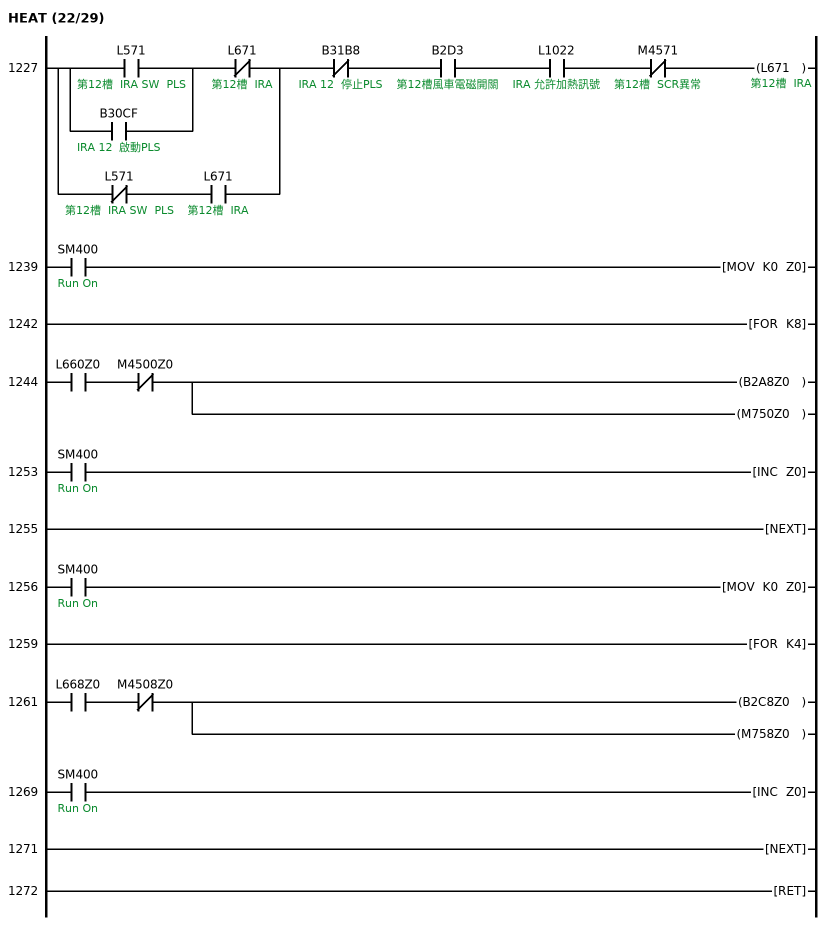
[picture p168: ladder of HEAT, rungs at steps 1227 to 1272]
1227  LD      L571  ; 第12槽  IRA SW  PLS
      OR      B30CF  ; IRA 12  啟動PLS
      ANI     L671  ; 第12槽  IRA
      LDI     L571  ; 第12槽  IRA SW  PLS
      AND     L671  ; 第12槽  IRA
      ORB
      ANI     B31B8  ; IRA 12  停止PLS
      AND     B2D3  ; 第12槽風車電磁開關
      AND     L1022  ; IRA 允許加熱訊號
      ANI     M4571  ; 第12槽  SCR異常
      OUT     L671  ; 第12槽  IRA
1239  LD      SM400  ; Run On
      MOV     K0 Z0
1242  FOR     K8
1244  LD      L660Z0
      ANI     M4500Z0
      OUT     B2A8Z0
      OUT     M750Z0
1253  LD      SM400  ; Run On
      INC     Z0
1255  NEXT
1256  LD      SM400  ; Run On
      MOV     K0 Z0
1259  FOR     K4
1261  LD      L668Z0
      ANI     M4508Z0
      OUT     B2C8Z0
      OUT     M758Z0
1269  LD      SM400  ; Run On
      INC     Z0
1271  NEXT
1272  RET
      P450
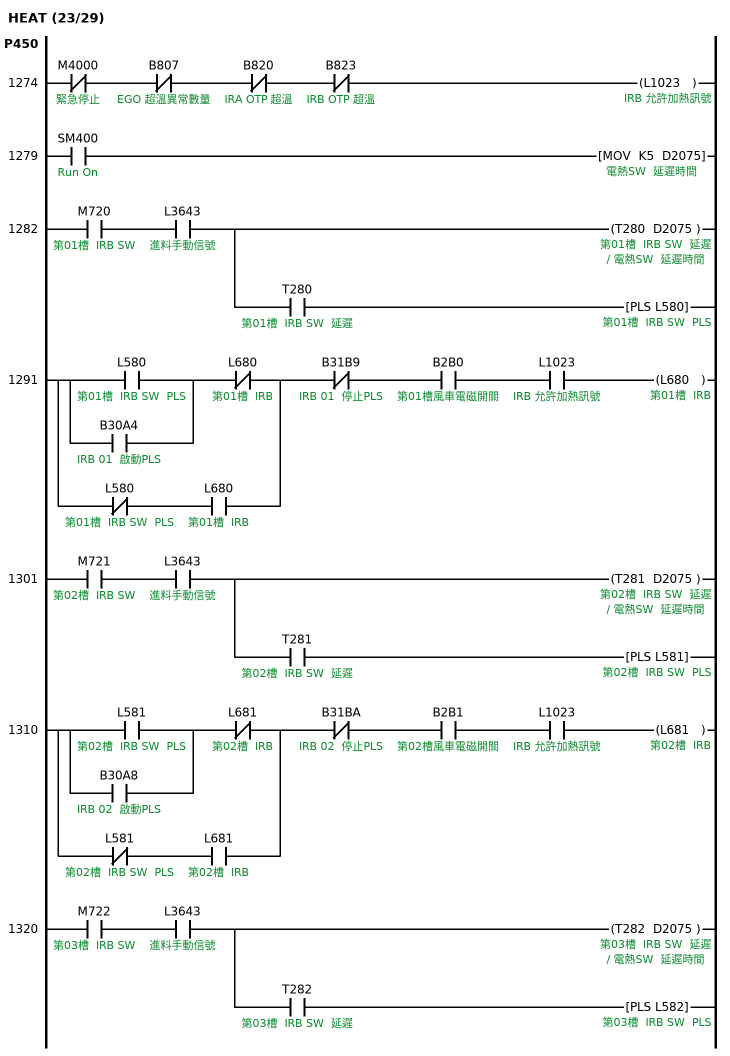
1274  LDI     M4000  ; 緊急停止
      ANI     B807  ; EGO 超溫異常數量
      ANI     B820  ; IRA OTP 超溫
      ANI     B823  ; IRB OTP 超溫
      OUT     L1023  ; IRB 允許加熱訊號
1279  LD      SM400  ; Run On
      MOV     K5 D2075
1282  LD      M720  ; 第01槽  IRB SW
      AND     L3643  ; 進料手動信號
      OUT     T280 D2075  ; 第01槽  IRB SW  延遲 / 電熱SW  延遲時間
      AND     T280  ; 第01槽  IRB SW  延遲
      PLS     L580  ; 第01槽  IRB SW  PLS
1291  LD      L580  ; 第01槽  IRB SW  PLS
      OR      B30A4  ; IRB 01  啟動PLS
      ANI     L680  ; 第01槽  IRB
      LDI     L580  ; 第01槽  IRB SW  PLS
      AND     L680  ; 第01槽  IRB
      ORB
      ANI     B31B9  ; IRB 01  停止PLS
      AND     B2B0  ; 第01槽風車電磁開關
      AND     L1023  ; IRB 允許加熱訊號
      OUT     L680  ; 第01槽  IRB
1301  LD      M721  ; 第02槽  IRB SW
      AND     L3643  ; 進料手動信號
      OUT     T281 D2075  ; 第02槽  IRB SW  延遲 / 電熱SW  延遲時間
      AND     T281  ; 第02槽  IRB SW  延遲
      PLS     L581  ; 第02槽  IRB SW  PLS
1310  LD      L581  ; 第02槽  IRB SW  PLS
      OR      B30A8  ; IRB 02  啟動PLS
      ANI     L681  ; 第02槽  IRB
      LDI     L581  ; 第02槽  IRB SW  PLS
      AND     L681  ; 第02槽  IRB
      ORB
      ANI     B31BA  ; IRB 02  停止PLS
      AND     B2B1  ; 第02槽風車電磁開關
      AND     L1023  ; IRB 允許加熱訊號
      OUT     L681  ; 第02槽  IRB
1320  LD      M722  ; 第03槽  IRB SW
      AND     L3643  ; 進料手動信號
      OUT     T282 D2075  ; 第03槽  IRB SW  延遲 / 電熱SW  延遲時間
      AND     T282  ; 第03槽  IRB SW  延遲
      PLS     L582  ; 第03槽  IRB SW  PLS
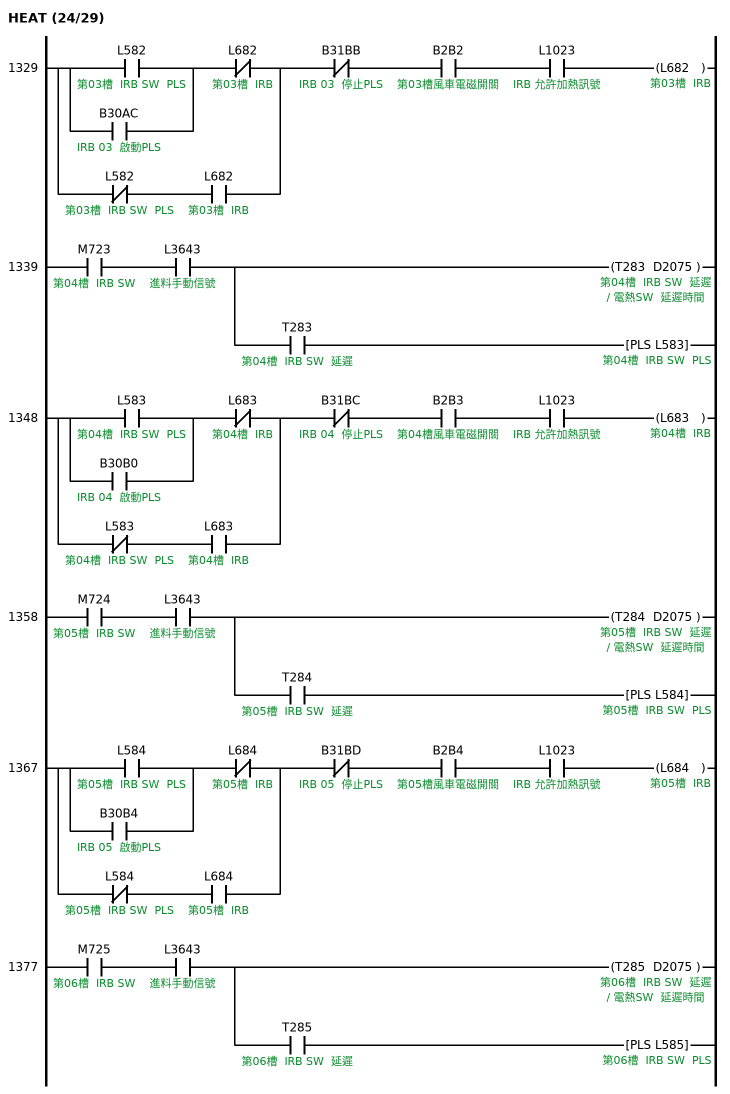
1329  LD      L582  ; 第03槽  IRB SW  PLS
      OR      B30AC  ; IRB 03  啟動PLS
      ANI     L682  ; 第03槽  IRB
      LDI     L582  ; 第03槽  IRB SW  PLS
      AND     L682  ; 第03槽  IRB
      ORB
      ANI     B31BB  ; IRB 03  停止PLS
      AND     B2B2  ; 第03槽風車電磁開關
      AND     L1023  ; IRB 允許加熱訊號
      OUT     L682  ; 第03槽  IRB
1339  LD      M723  ; 第04槽  IRB SW
      AND     L3643  ; 進料手動信號
      OUT     T283 D2075  ; 第04槽  IRB SW  延遲 / 電熱SW  延遲時間
      AND     T283  ; 第04槽  IRB SW  延遲
      PLS     L583  ; 第04槽  IRB SW  PLS
1348  LD      L583  ; 第04槽  IRB SW  PLS
      OR      B30B0  ; IRB 04  啟動PLS
      ANI     L683  ; 第04槽  IRB
      LDI     L583  ; 第04槽  IRB SW  PLS
      AND     L683  ; 第04槽  IRB
      ORB
      ANI     B31BC  ; IRB 04  停止PLS
      AND     B2B3  ; 第04槽風車電磁開關
      AND     L1023  ; IRB 允許加熱訊號
      OUT     L683  ; 第04槽  IRB
1358  LD      M724  ; 第05槽  IRB SW
      AND     L3643  ; 進料手動信號
      OUT     T284 D2075  ; 第05槽  IRB SW  延遲 / 電熱SW  延遲時間
      AND     T284  ; 第05槽  IRB SW  延遲
      PLS     L584  ; 第05槽  IRB SW  PLS
1367  LD      L584  ; 第05槽  IRB SW  PLS
      OR      B30B4  ; IRB 05  啟動PLS
      ANI     L684  ; 第05槽  IRB
      LDI     L584  ; 第05槽  IRB SW  PLS
      AND     L684  ; 第05槽  IRB
      ORB
      ANI     B31BD  ; IRB 05  停止PLS
      AND     B2B4  ; 第05槽風車電磁開關
      AND     L1023  ; IRB 允許加熱訊號
      OUT     L684  ; 第05槽  IRB
1377  LD      M725  ; 第06槽  IRB SW
      AND     L3643  ; 進料手動信號
      OUT     T285 D2075  ; 第06槽  IRB SW  延遲 / 電熱SW  延遲時間
      AND     T285  ; 第06槽  IRB SW  延遲
      PLS     L585  ; 第06槽  IRB SW  PLS
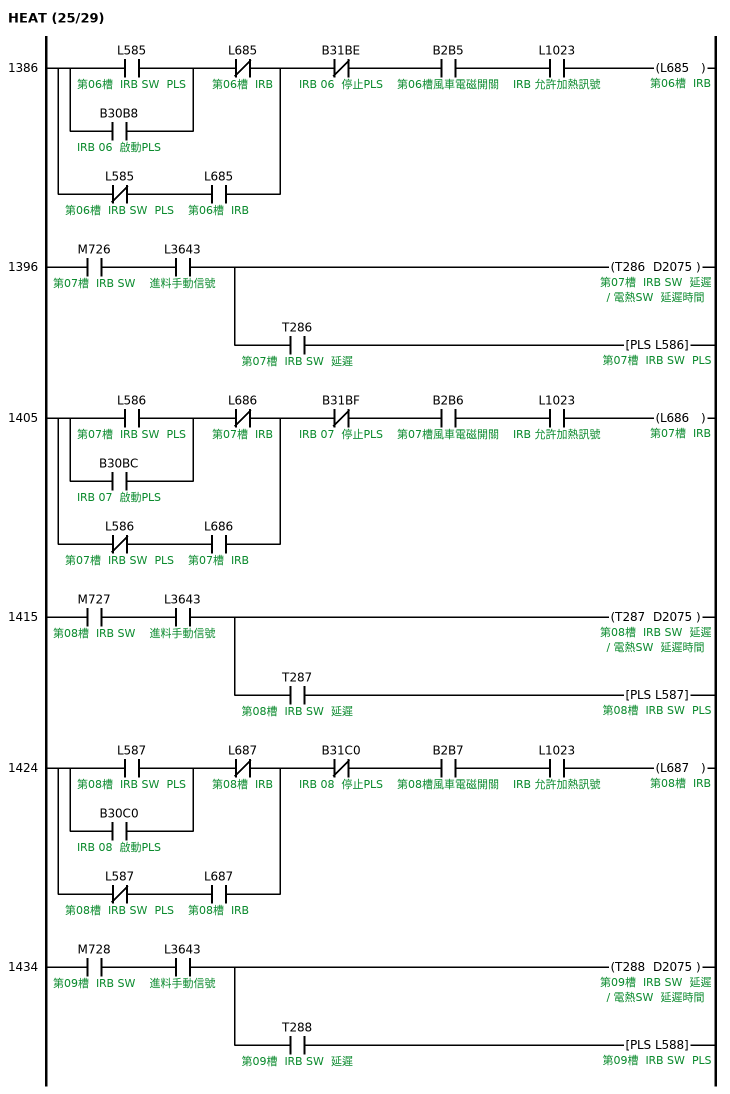
1386  LD      L585  ; 第06槽  IRB SW  PLS
      OR      B30B8  ; IRB 06  啟動PLS
      ANI     L685  ; 第06槽  IRB
      LDI     L585  ; 第06槽  IRB SW  PLS
      AND     L685  ; 第06槽  IRB
      ORB
      ANI     B31BE  ; IRB 06  停止PLS
      AND     B2B5  ; 第06槽風車電磁開關
      AND     L1023  ; IRB 允許加熱訊號
      OUT     L685  ; 第06槽  IRB
1396  LD      M726  ; 第07槽  IRB SW
      AND     L3643  ; 進料手動信號
      OUT     T286 D2075  ; 第07槽  IRB SW  延遲 / 電熱SW  延遲時間
      AND     T286  ; 第07槽  IRB SW  延遲
      PLS     L586  ; 第07槽  IRB SW  PLS
1405  LD      L586  ; 第07槽  IRB SW  PLS
      OR      B30BC  ; IRB 07  啟動PLS
      ANI     L686  ; 第07槽  IRB
      LDI     L586  ; 第07槽  IRB SW  PLS
      AND     L686  ; 第07槽  IRB
      ORB
      ANI     B31BF  ; IRB 07  停止PLS
      AND     B2B6  ; 第07槽風車電磁開關
      AND     L1023  ; IRB 允許加熱訊號
      OUT     L686  ; 第07槽  IRB
1415  LD      M727  ; 第08槽  IRB SW
      AND     L3643  ; 進料手動信號
      OUT     T287 D2075  ; 第08槽  IRB SW  延遲 / 電熱SW  延遲時間
      AND     T287  ; 第08槽  IRB SW  延遲
      PLS     L587  ; 第08槽  IRB SW  PLS
1424  LD      L587  ; 第08槽  IRB SW  PLS
      OR      B30C0  ; IRB 08  啟動PLS
      ANI     L687  ; 第08槽  IRB
      LDI     L587  ; 第08槽  IRB SW  PLS
      AND     L687  ; 第08槽  IRB
      ORB
      ANI     B31C0  ; IRB 08  停止PLS
      AND     B2B7  ; 第08槽風車電磁開關
      AND     L1023  ; IRB 允許加熱訊號
      OUT     L687  ; 第08槽  IRB
1434  LD      M728  ; 第09槽  IRB SW
      AND     L3643  ; 進料手動信號
      OUT     T288 D2075  ; 第09槽  IRB SW  延遲 / 電熱SW  延遲時間
      AND     T288  ; 第09槽  IRB SW  延遲
      PLS     L588  ; 第09槽  IRB SW  PLS
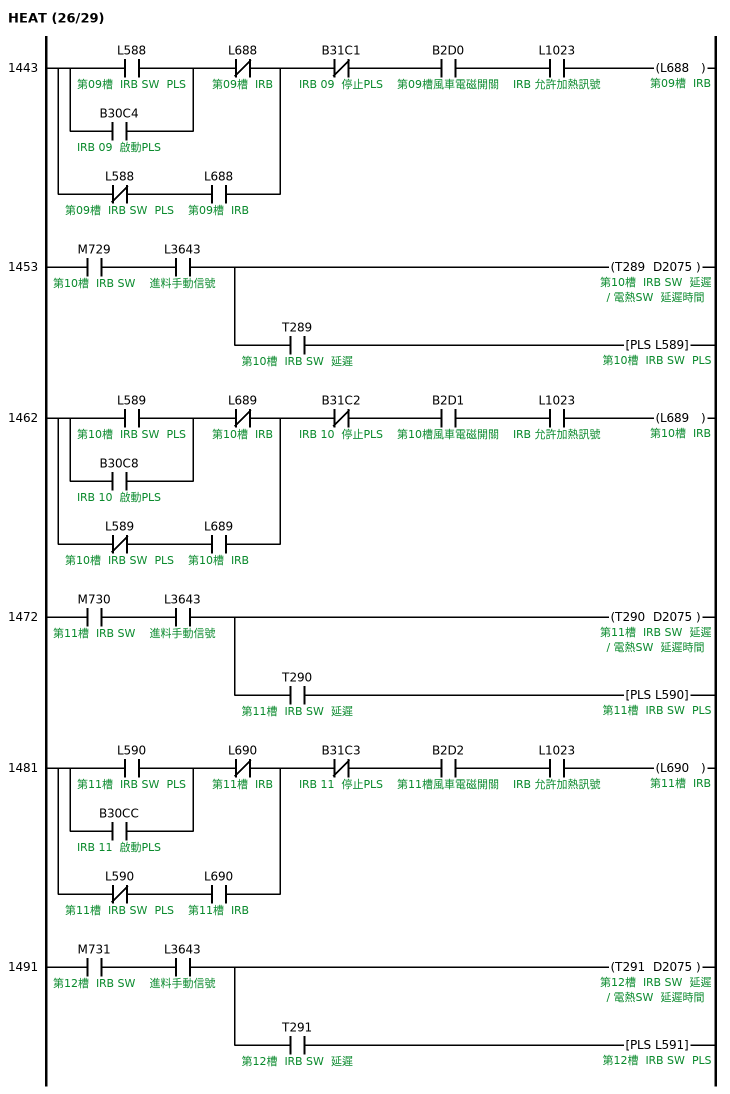
1443  LD      L588  ; 第09槽  IRB SW  PLS
      OR      B30C4  ; IRB 09  啟動PLS
      ANI     L688  ; 第09槽  IRB
      LDI     L588  ; 第09槽  IRB SW  PLS
      AND     L688  ; 第09槽  IRB
      ORB
      ANI     B31C1  ; IRB 09  停止PLS
      AND     B2D0  ; 第09槽風車電磁開關
      AND     L1023  ; IRB 允許加熱訊號
      OUT     L688  ; 第09槽  IRB
1453  LD      M729  ; 第10槽  IRB SW
      AND     L3643  ; 進料手動信號
      OUT     T289 D2075  ; 第10槽  IRB SW  延遲 / 電熱SW  延遲時間
      AND     T289  ; 第10槽  IRB SW  延遲
      PLS     L589  ; 第10槽  IRB SW  PLS
1462  LD      L589  ; 第10槽  IRB SW  PLS
      OR      B30C8  ; IRB 10  啟動PLS
      ANI     L689  ; 第10槽  IRB
      LDI     L589  ; 第10槽  IRB SW  PLS
      AND     L689  ; 第10槽  IRB
      ORB
      ANI     B31C2  ; IRB 10  停止PLS
      AND     B2D1  ; 第10槽風車電磁開關
      AND     L1023  ; IRB 允許加熱訊號
      OUT     L689  ; 第10槽  IRB
1472  LD      M730  ; 第11槽  IRB SW
      AND     L3643  ; 進料手動信號
      OUT     T290 D2075  ; 第11槽  IRB SW  延遲 / 電熱SW  延遲時間
      AND     T290  ; 第11槽  IRB SW  延遲
      PLS     L590  ; 第11槽  IRB SW  PLS
1481  LD      L590  ; 第11槽  IRB SW  PLS
      OR      B30CC  ; IRB 11  啟動PLS
      ANI     L690  ; 第11槽  IRB
      LDI     L590  ; 第11槽  IRB SW  PLS
      AND     L690  ; 第11槽  IRB
      ORB
      ANI     B31C3  ; IRB 11  停止PLS
      AND     B2D2  ; 第11槽風車電磁開關
      AND     L1023  ; IRB 允許加熱訊號
      OUT     L690  ; 第11槽  IRB
1491  LD      M731  ; 第12槽  IRB SW
      AND     L3643  ; 進料手動信號
      OUT     T291 D2075  ; 第12槽  IRB SW  延遲 / 電熱SW  延遲時間
      AND     T291  ; 第12槽  IRB SW  延遲
      PLS     L591  ; 第12槽  IRB SW  PLS
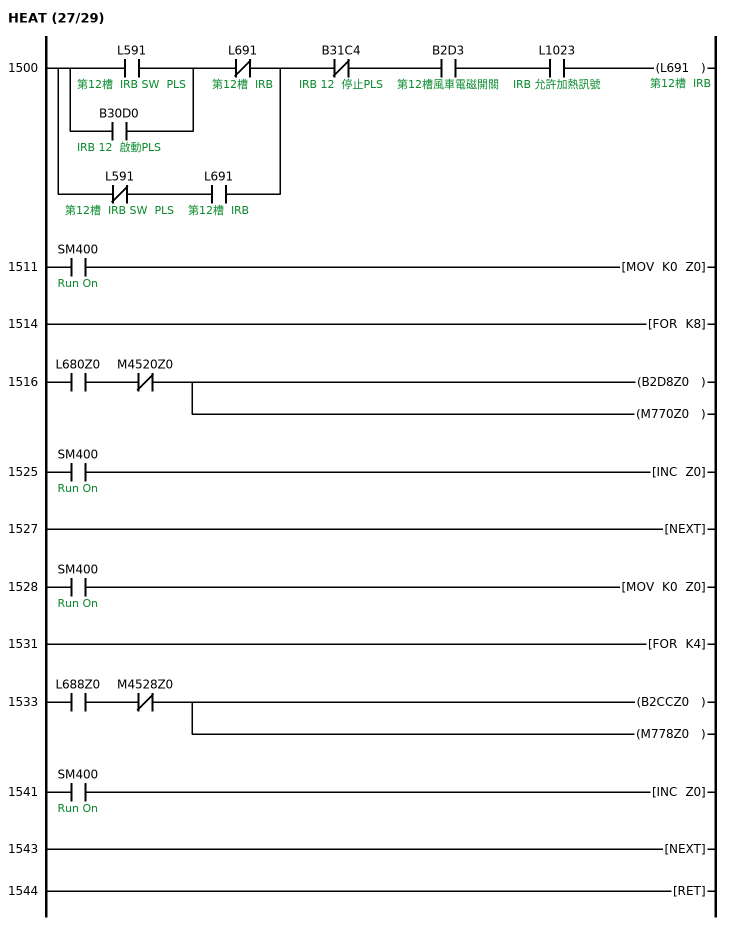
1500  LD      L591  ; 第12槽  IRB SW  PLS
      OR      B30D0  ; IRB 12  啟動PLS
      ANI     L691  ; 第12槽  IRB
      LDI     L591  ; 第12槽  IRB SW  PLS
      AND     L691  ; 第12槽  IRB
      ORB
      ANI     B31C4  ; IRB 12  停止PLS
      AND     B2D3  ; 第12槽風車電磁開關
      AND     L1023  ; IRB 允許加熱訊號
      OUT     L691  ; 第12槽  IRB
1511  LD      SM400  ; Run On
      MOV     K0 Z0
1514  FOR     K8
1516  LD      L680Z0
      ANI     M4520Z0
      OUT     B2D8Z0
      OUT     M770Z0
1525  LD      SM400  ; Run On
      INC     Z0
1527  NEXT
1528  LD      SM400  ; Run On
      MOV     K0 Z0
1531  FOR     K4
1533  LD      L688Z0
      ANI     M4528Z0
      OUT     B2CCZ0
      OUT     M778Z0
1541  LD      SM400  ; Run On
      INC     Z0
1543  NEXT
1544  RET
; /* Length=每段爐體長度_Section=爐體段數 */
      P460
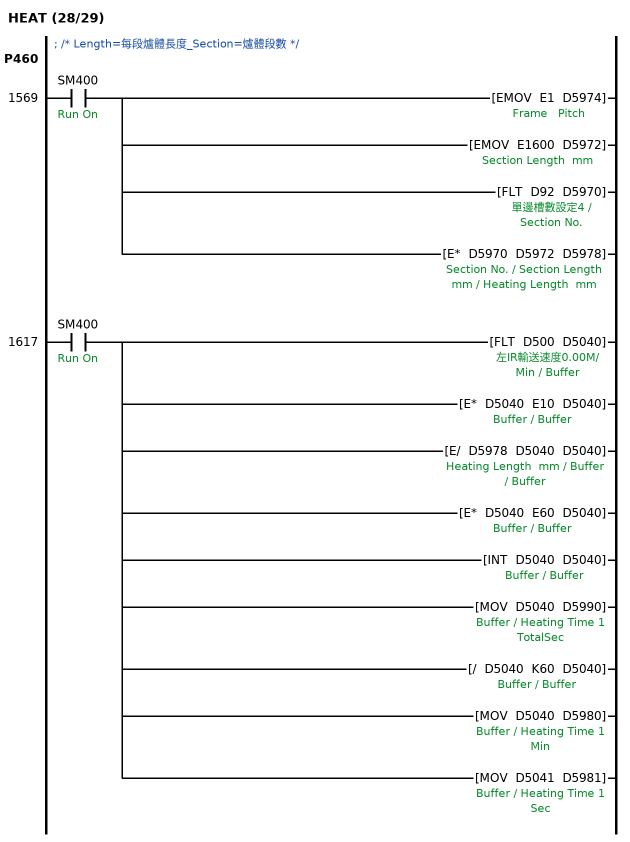
1569  LD      SM400  ; Run On
      EMOV    E1 D5974  ; Frame   Pitch
      EMOV    E1600 D5972  ; Section Length  mm
        [note] /* 加熱爐體每段長度mm */
      FLT     D92 D5970  ; 單邊槽數設定4 / Section No.
        [note] /* 加熱段數 */
      E*      D5970 D5972 D5978  ; Heating Length  mm
        [note] /* 加熱段_總長度mm */
1617  LD      SM400  ; Run On
      FLT     D500 D5040  ; 左IR輸送速度0.00M/Min / Buffer
      E*      D5040 E10 D5040
      E/      D5978 D5040 D5040
        [note] / 板子經過爐體總時間_E0.000Min /
      E*      D5040 E60 D5040
        [note] / 板子經過爐體總時間_E0.000Sec /
      INT     D5040 D5040
      MOV     D5040 D5990  ; Heating Time 1  TotalSec
      /       D5040 K60 D5040
      MOV     D5040 D5980  ; Heating Time 1  Min
      MOV     D5041 D5981  ; Buffer / Heating Time 1  Sec
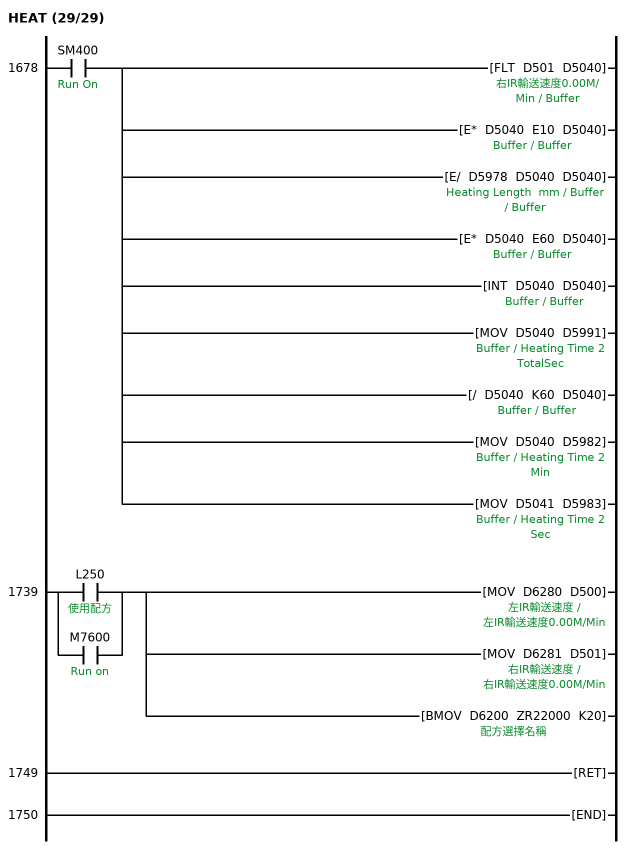
1678  LD      SM400  ; Run On
      FLT     D501 D5040  ; 右IR輸送速度0.00M/Min
      E*      D5040 E10 D5040
      E/      D5978 D5040 D5040
        [note] / 板子經過爐體總時間_E0.000Min /
      E*      D5040 E60 D5040
        [note] / 板子經過爐體總時間_E0.000Sec /
      INT     D5040 D5040
      MOV     D5040 D5991  ; Heating Time 2  TotalSec
      /       D5040 K60 D5040
      MOV     D5040 D5982  ; Heating Time 2  Min
      MOV     D5041 D5983  ; Heating Time 2  Sec
1739  LD      L250  ; 使用配方
      OR      M7600  ; Run on
      MOV     D6280 D500  ; 左IR輸送速度
      MOV     D6281 D501  ; 右IR輸送速度
      BMOV    D6200 ZR22000 K20  ; 配方選擇名稱
1749  RET
1750  END
END_PROGRAM

PROGRAM ALARM
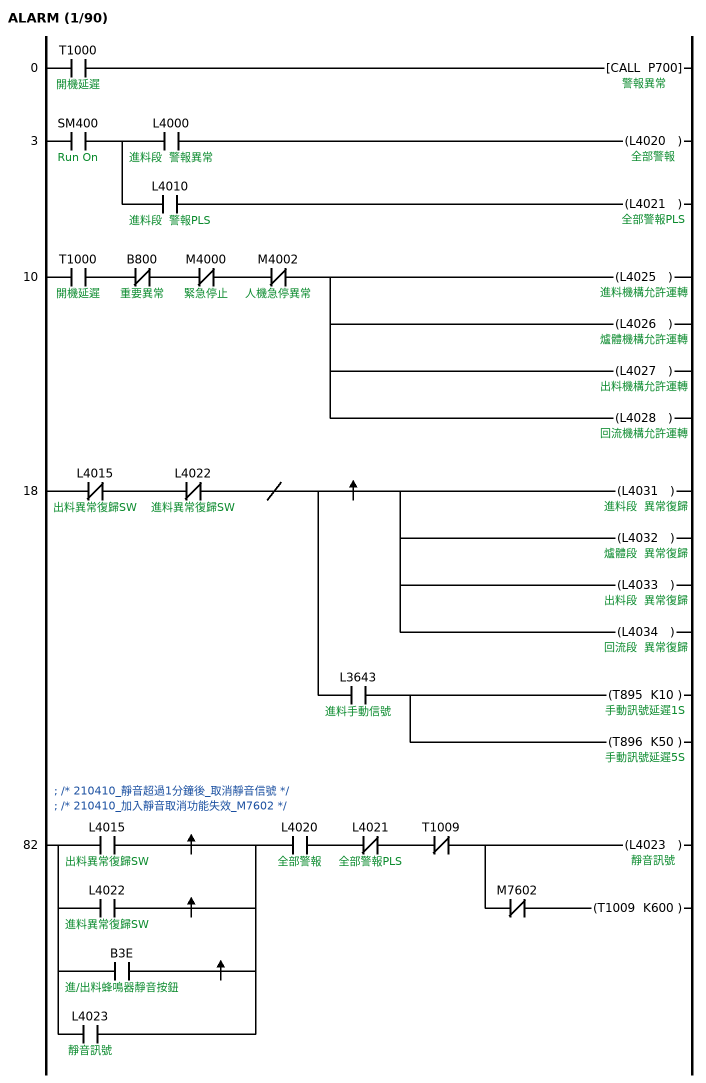
0     LD      T1000  ; 開機延遲
      CALL    P700  ; 警報異常
3     LD      SM400  ; Run On
      MPS
      AND     L4000  ; 進料段  警報異常
      OUT     L4020  ; 全部警報
      MPP
      AND     L4010  ; 進料段  警報PLS
      OUT     L4021  ; 全部警報PLS
10    LD      T1000  ; 開機延遲
      ANI     B800  ; 重要異常
      ANI     M4000  ; 緊急停止
      ANI     M4002  ; 人機急停異常
      OUT     L4025  ; 進料機構允許運轉
      OUT     L4026  ; 爐體機構允許運轉
      OUT     L4027  ; 出料機構允許運轉
      OUT     L4028  ; 回流機構允許運轉
18    LDI     L4015  ; 出料異常復歸SW
      ANI     L4022  ; 進料異常復歸SW
      INV
      MPS
      MEP
      OUT     L4031  ; 進料段  異常復歸
      OUT     L4032  ; 爐體段  異常復歸
      OUT     L4033  ; 出料段  異常復歸
      OUT     L4034  ; 回流段  異常復歸
      MPP
      AND     L3643  ; 進料手動信號
      OUT     T895 K10  ; 手動訊號延遲1S
      OUT     T896 K50  ; 手動訊號延遲5S
; /* 210410_靜音超過1分鐘後_取消靜音信號 */
; /* 210410_加入靜音取消功能失效_M7602 */
82    LD      L4015  ; 出料異常復歸SW
      MEP
      LD      L4022  ; 進料異常復歸SW
      MEP
      ORB
      LD      B3E  ; 進/出料蜂鳴器靜音按鈕
      MEP
      ORB
      OR      L4023  ; 靜音訊號
      AND     L4020  ; 全部警報
      ANI     L4021  ; 全部警報PLS
      ANI     T1009
      OUT     L4023  ; 靜音訊號
      ANI     M7602
      OUT     T1009 K600
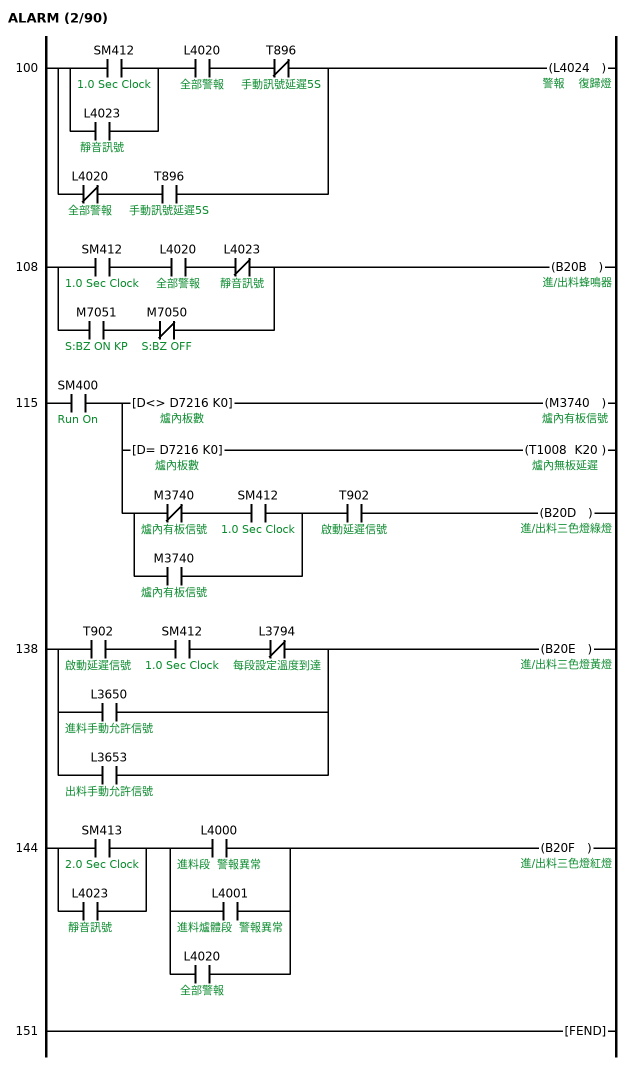
100   LD      SM412  ; 1.0 Sec Clock
      OR      L4023  ; 靜音訊號
      AND     L4020  ; 全部警報
      ANI     T896  ; 手動訊號延遲5S
      LDI     L4020  ; 全部警報
      AND     T896  ; 手動訊號延遲5S
      ORB
      OUT     L4024  ; 警報    復歸燈
108   LD      SM412  ; 1.0 Sec Clock
      AND     L4020  ; 全部警報
      ANI     L4023  ; 靜音訊號
      LD      M7051  ; S:BZ ON KP
      ANI     M7050  ; S:BZ OFF
      ORB
      OUT     B20B  ; 進/出料蜂鳴器
115   LD      SM400  ; Run On
      MPS
      ANDD<>  D7216 K0  ; 爐內板數
      OUT     M3740  ; 爐內有板信號
      MRD
      ANDD=   D7216 K0  ; 爐內板數
      OUT     T1008 K20  ; 爐內無板延遲
      MPP
      LDI     M3740  ; 爐內有板信號
      AND     SM412  ; 1.0 Sec Clock
      OR      M3740  ; 爐內有板信號
      ANB
      AND     T902  ; 啟動延遲信號
      OUT     B20D  ; 進/出料三色燈綠燈
138   LD      T902  ; 啟動延遲信號
      AND     SM412  ; 1.0 Sec Clock
      ANI     L3794  ; 每段設定溫度到達
      OR      L3650  ; 進料手動允許信號
      OR      L3653  ; 出料手動允許信號
      OUT     B20E  ; 進/出料三色燈黃燈
144   LD      SM413  ; 2.0 Sec Clock
      OR      L4023  ; 靜音訊號
      LD      L4000  ; 進料段  警報異常
      OR      L4001  ; 進料爐體段  警報異常
      OR      L4020  ; 全部警報
      ANB
      OUT     B20F  ; 進/出料三色燈紅燈
151   FEND
      P700
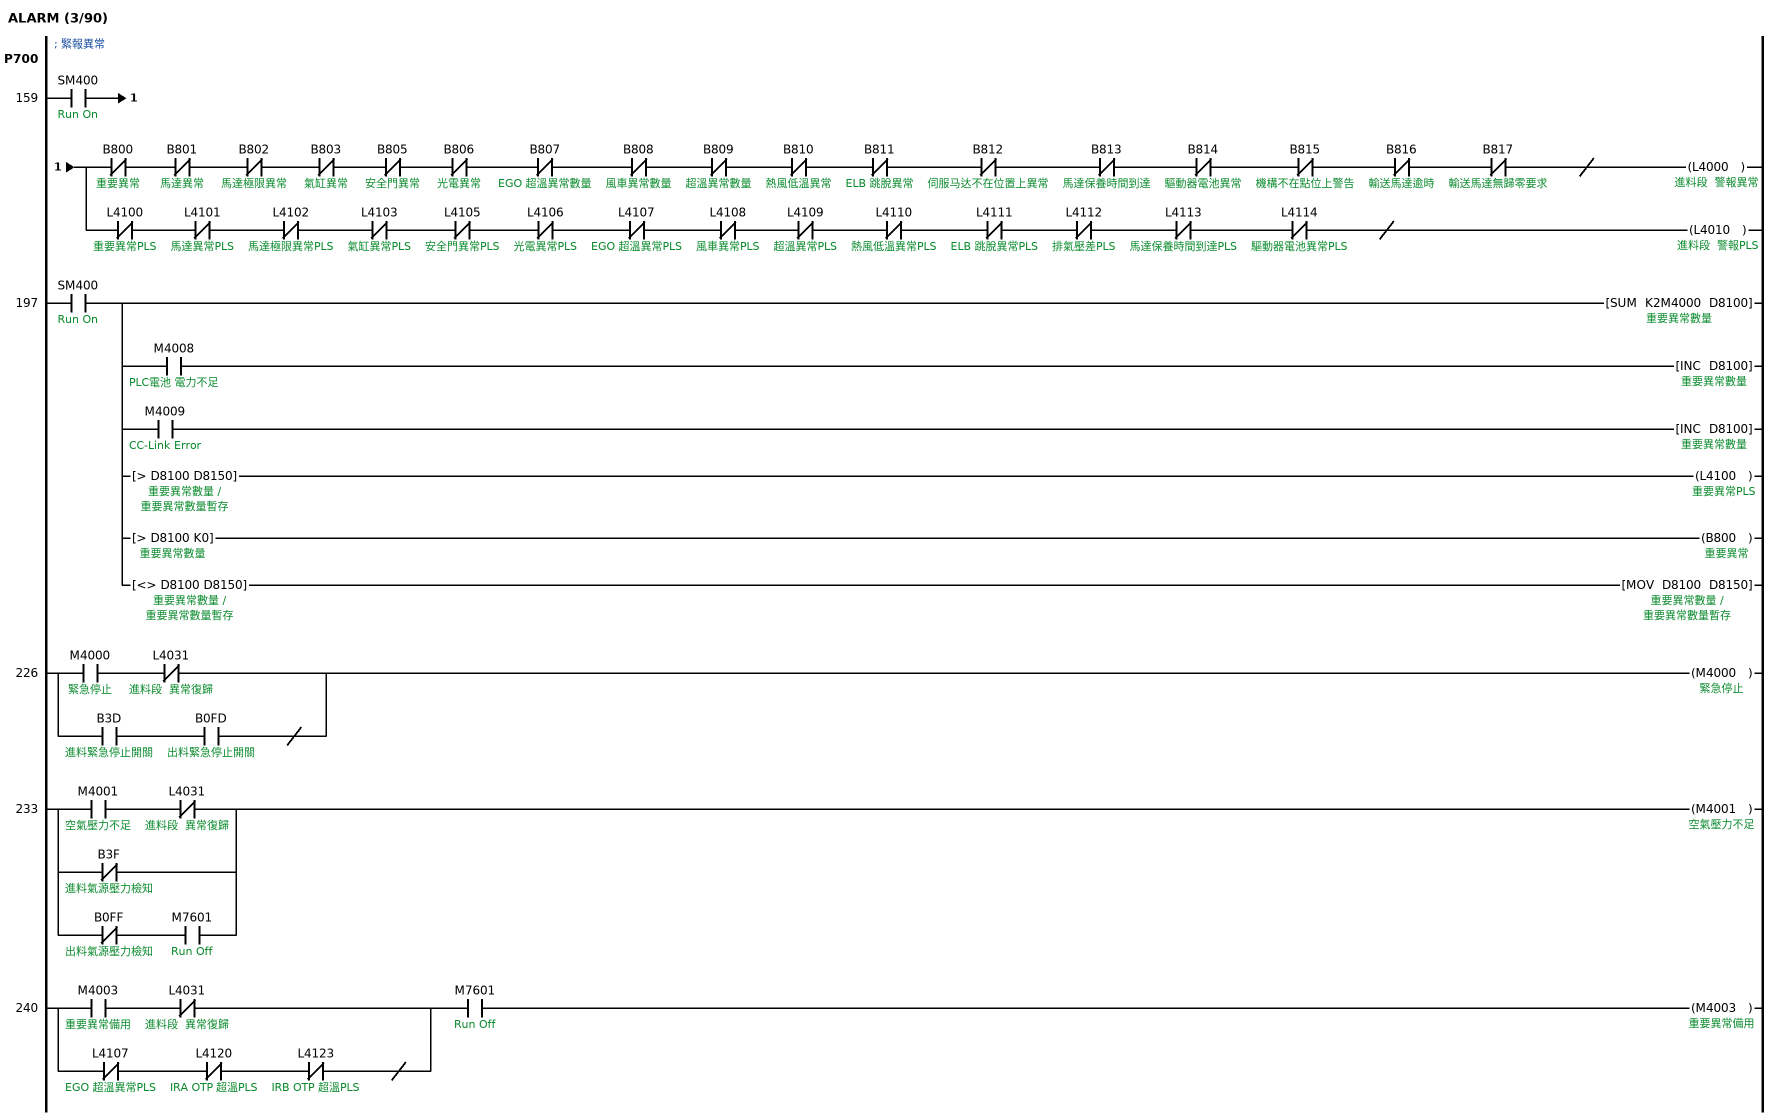
; 緊報異常
159   LD      SM400  ; Run On
      MPS
      ANI     B800  ; 重要異常
      ANI     B801  ; 馬達異常
      ANI     B802  ; 馬達極限異常
      ANI     B803  ; 氣缸異常
      ANI     B805  ; 安全門異常
      ANI     B806  ; 光電異常
      ANI     B807  ; EGO 超溫異常數量
      ANI     B808  ; 風車異常數量
      ANI     B809  ; 超溫異常數量
      ANI     B810  ; 熱風低溫異常
      ANI     B811  ; ELB 跳脫異常
      ANI     B812  ; 伺服马达不在位置上異常
      ANI     B813  ; 馬達保養時間到達
      ANI     B814  ; 驅動器電池異常
      ANI     B815  ; 機構不在點位上警告
      ANI     B816  ; 輸送馬達逾時
      ANI     B817  ; 輸送馬達無歸零要求
      INV
      OUT     L4000  ; 進料段  警報異常
      MPP
      ANI     L4100  ; 重要異常PLS
      ANI     L4101  ; 馬達異常PLS
      ANI     L4102  ; 馬達極限異常PLS
      ANI     L4103  ; 氣缸異常PLS
      ANI     L4105  ; 安全門異常PLS
      ANI     L4106  ; 光電異常PLS
      ANI     L4107  ; EGO 超溫異常PLS
      ANI     L4108  ; 風車異常PLS
      ANI     L4109  ; 超溫異常PLS
      ANI     L4110  ; 熱風低溫異常PLS
      ANI     L4111  ; ELB 跳脫異常PLS
      ANI     L4112  ; 排氣壓差PLS
      ANI     L4113  ; 馬達保養時間到達PLS
      ANI     L4114  ; 驅動器電池異常PLS
      INV
      OUT     L4010  ; 進料段  警報PLS
197   LD      SM400  ; Run On
      SUM     K2M4000 D8100  ; 重要異常數量
      MPS
      AND     M4008  ; PLC電池 電力不足
      INC     D8100
      MRD
      AND     M4009  ; CC-Link Error
      INC     D8100
      MRD
      AND>    D8100 D8150  ; 重要異常數量 / 重要異常數量暫存
      OUT     L4100  ; 重要異常PLS
      MRD
      AND>    D8100 K0  ; 重要異常數量
      OUT     B800  ; 重要異常
      MPP
      AND<>   D8100 D8150  ; 重要異常數量 / 重要異常數量暫存
      MOV     D8100 D8150
226   LD      M4000  ; 緊急停止
      ANI     L4031  ; 進料段  異常復歸
      LD      B3D  ; 進料緊急停止開關
      AND     B0FD  ; 出料緊急停止開關
      INV
      ORB
      OUT     M4000  ; 緊急停止
233   LD      M4001  ; 空氣壓力不足
      ANI     L4031  ; 進料段  異常復歸
      ORI     B3F  ; 進料氣源壓力檢知
      LDI     B0FF  ; 出料氣源壓力檢知
      AND     M7601  ; Run Off
      ORB
      OUT     M4001  ; 空氣壓力不足
240   LD      M4003  ; 重要異常備用
      ANI     L4031  ; 進料段  異常復歸
      LDI     L4107  ; EGO 超溫異常PLS
      ANI     L4120  ; IRA OTP 超溫PLS
      ANI     L4123  ; IRB OTP 超溫PLS
      INV
      ORB
      AND     M7601  ; Run Off
      OUT     M4003  ; 重要異常備用
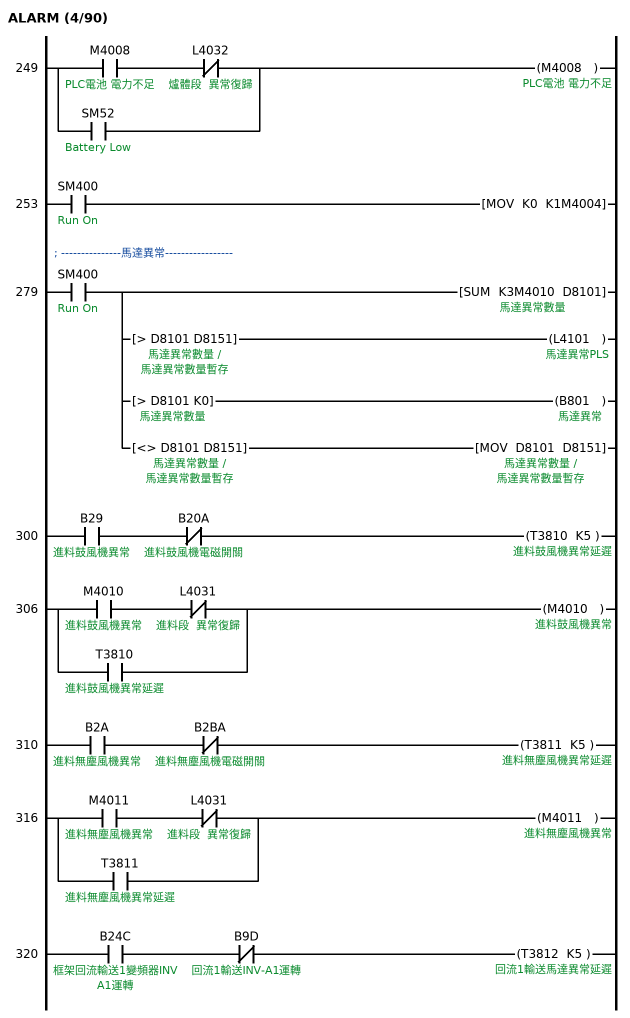
249   LD      M4008  ; PLC電池 電力不足
      ANI     L4032  ; 爐體段  異常復歸
      OR      SM52  ; Battery Low
      OUT     M4008  ; PLC電池 電力不足
253   LD      SM400  ; Run On
      MOV     K0 K1M4004  ; 重要異常備用
; ---------------馬達異常-----------------
279   LD      SM400  ; Run On
      SUM     K3M4010 D8101  ; 進料鼓風機異常 / 馬達異常數量
      MPS
      AND>    D8101 D8151  ; 馬達異常數量 / 馬達異常數量暫存
      OUT     L4101  ; 馬達異常PLS
      MRD
      AND>    D8101 K0  ; 馬達異常數量
      OUT     B801  ; 馬達異常
      MPP
      AND<>   D8101 D8151  ; 馬達異常數量 / 馬達異常數量暫存
      MOV     D8101 D8151
300   LD      B29  ; 進料鼓風機異常
      ANI     B20A  ; 進料鼓風機電磁開關
      OUT     T3810 K5  ; 進料鼓風機異常延遲
306   LD      M4010  ; 進料鼓風機異常
      ANI     L4031  ; 進料段  異常復歸
      OR      T3810  ; 進料鼓風機異常延遲
      OUT     M4010  ; 進料鼓風機異常
310   LD      B2A  ; 進料無塵風機異常
      ANI     B2BA  ; 進料無塵風機電磁開關
      OUT     T3811 K5  ; 進料無塵風機異常延遲
316   LD      M4011  ; 進料無塵風機異常
      ANI     L4031  ; 進料段  異常復歸
      OR      T3811  ; 進料無塵風機異常延遲
      OUT     M4011  ; 進料無塵風機異常
320   LD      B24C  ; 框架回流輸送1變頻器INVA1運轉
      ANI     B9D  ; 回流1輸送INV-A1運轉
      OUT     T3812 K5  ; 回流1輸送馬達異常延遲
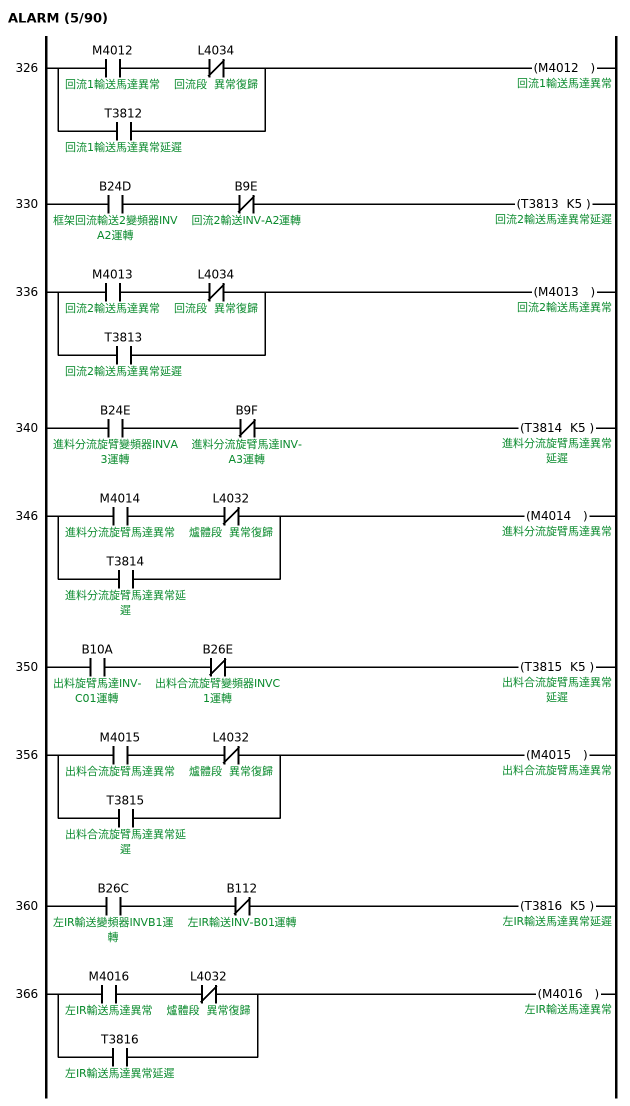
326   LD      M4012  ; 回流1輸送馬達異常
      ANI     L4034  ; 回流段  異常復歸
      OR      T3812  ; 回流1輸送馬達異常延遲
      OUT     M4012  ; 回流1輸送馬達異常
330   LD      B24D  ; 框架回流輸送2變頻器INVA2運轉
      ANI     B9E  ; 回流2輸送INV-A2運轉
      OUT     T3813 K5  ; 回流2輸送馬達異常延遲
336   LD      M4013  ; 回流2輸送馬達異常
      ANI     L4034  ; 回流段  異常復歸
      OR      T3813  ; 回流2輸送馬達異常延遲
      OUT     M4013  ; 回流2輸送馬達異常
340   LD      B24E  ; 進料分流旋臂變頻器INVA3運轉
      ANI     B9F  ; 進料分流旋臂馬達INV-A3運轉
      OUT     T3814 K5  ; 進料分流旋臂馬達異常延遲
346   LD      M4014  ; 進料分流旋臂馬達異常
      ANI     L4032  ; 爐體段  異常復歸
      OR      T3814  ; 進料分流旋臂馬達異常延遲
      OUT     M4014  ; 進料分流旋臂馬達異常
350   LD      B10A  ; 出料旋臂馬達INV-C01運轉
      ANI     B26E  ; 出料合流旋臂變頻器INVC1運轉
      OUT     T3815 K5  ; 出料合流旋臂馬達異常延遲
356   LD      M4015  ; 出料合流旋臂馬達異常
      ANI     L4032  ; 爐體段  異常復歸
      OR      T3815  ; 出料合流旋臂馬達異常延遲
      OUT     M4015  ; 出料合流旋臂馬達異常
360   LD      B26C  ; 左IR輸送變頻器INVB1運轉
      ANI     B112  ; 左IR輸送INV-B01運轉
      OUT     T3816 K5  ; 左IR輸送馬達異常延遲
366   LD      M4016  ; 左IR輸送馬達異常
      ANI     L4032  ; 爐體段  異常復歸
      OR      T3816  ; 左IR輸送馬達異常延遲
      OUT     M4016  ; 左IR輸送馬達異常
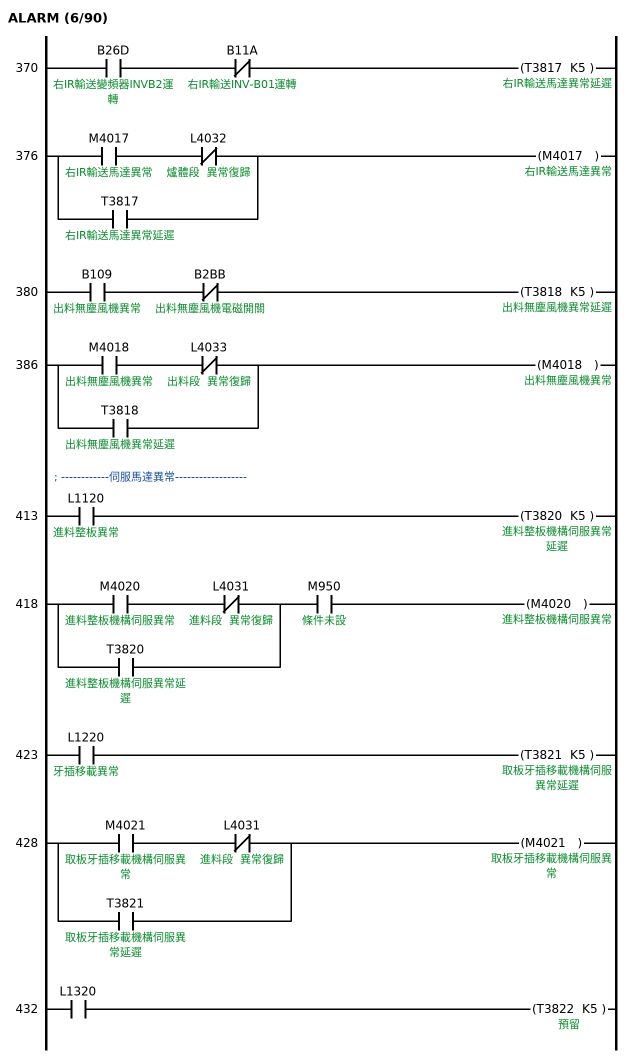
370   LD      B26D  ; 右IR輸送變頻器INVB2運轉
      ANI     B11A  ; 右IR輸送INV-B01運轉
      OUT     T3817 K5  ; 右IR輸送馬達異常延遲
376   LD      M4017  ; 右IR輸送馬達異常
      ANI     L4032  ; 爐體段  異常復歸
      OR      T3817  ; 右IR輸送馬達異常延遲
      OUT     M4017  ; 右IR輸送馬達異常
380   LD      B109  ; 出料無塵風機異常
      ANI     B2BB  ; 出料無塵風機電磁開關
      OUT     T3818 K5  ; 出料無塵風機異常延遲
386   LD      M4018  ; 出料無塵風機異常
      ANI     L4033  ; 出料段  異常復歸
      OR      T3818  ; 出料無塵風機異常延遲
      OUT     M4018  ; 出料無塵風機異常
; ------------伺服馬達異常------------------
413   LD      L1120  ; 進料整板異常
      OUT     T3820 K5  ; 進料整板機構伺服異常延遲
418   LD      M4020  ; 進料整板機構伺服異常
      ANI     L4031  ; 進料段  異常復歸
      OR      T3820  ; 進料整板機構伺服異常延遲
      AND     M950  ; 條件未設
      OUT     M4020  ; 進料整板機構伺服異常
423   LD      L1220  ; 牙插移載異常
      OUT     T3821 K5  ; 取板牙插移載機構伺服異常延遲
428   LD      M4021  ; 取板牙插移載機構伺服異常
      ANI     L4031  ; 進料段  異常復歸
      OR      T3821  ; 取板牙插移載機構伺服異常延遲
      OUT     M4021  ; 取板牙插移載機構伺服異常
432   LD      L1320
      OUT     T3822 K5  ; 預留
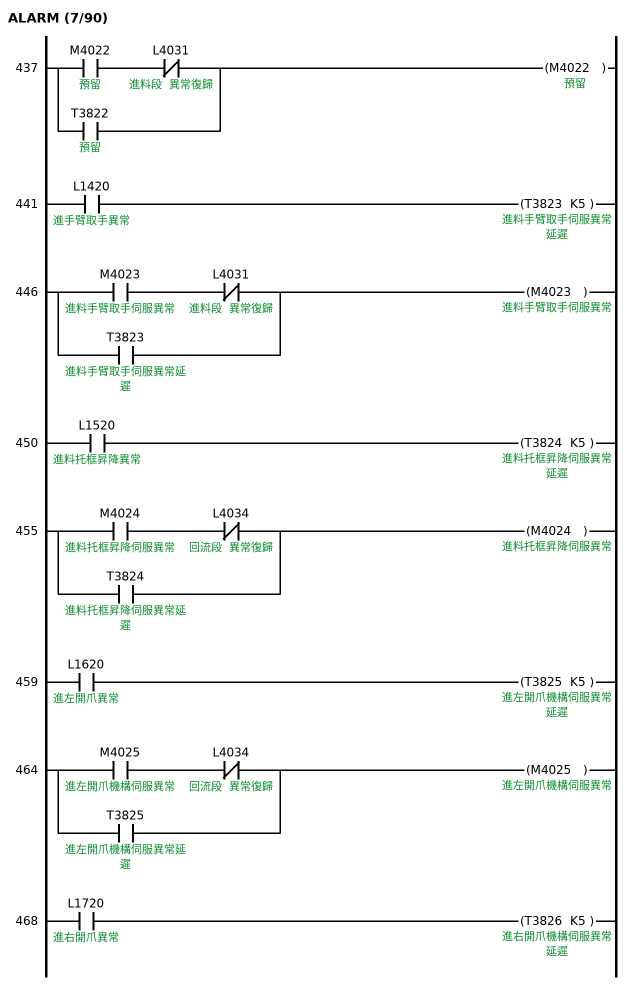
437   LD      M4022  ; 預留
      ANI     L4031  ; 進料段  異常復歸
      OR      T3822  ; 預留
      OUT     M4022  ; 預留
441   LD      L1420  ; 進手臂取手異常
      OUT     T3823 K5  ; 進料手臂取手伺服異常延遲
446   LD      M4023  ; 進料手臂取手伺服異常
      ANI     L4031  ; 進料段  異常復歸
      OR      T3823  ; 進料手臂取手伺服異常延遲
      OUT     M4023  ; 進料手臂取手伺服異常
450   LD      L1520  ; 進料托框昇降異常
      OUT     T3824 K5  ; 進料托框昇降伺服異常延遲
455   LD      M4024  ; 進料托框昇降伺服異常
      ANI     L4034  ; 回流段  異常復歸
      OR      T3824  ; 進料托框昇降伺服異常延遲
      OUT     M4024  ; 進料托框昇降伺服異常
459   LD      L1620  ; 進左開爪異常
      OUT     T3825 K5  ; 進左開爪機構伺服異常延遲
464   LD      M4025  ; 進左開爪機構伺服異常
      ANI     L4034  ; 回流段  異常復歸
      OR      T3825  ; 進左開爪機構伺服異常延遲
      OUT     M4025  ; 進左開爪機構伺服異常
468   LD      L1720  ; 進右開爪異常
      OUT     T3826 K5  ; 進右開爪機構伺服異常延遲
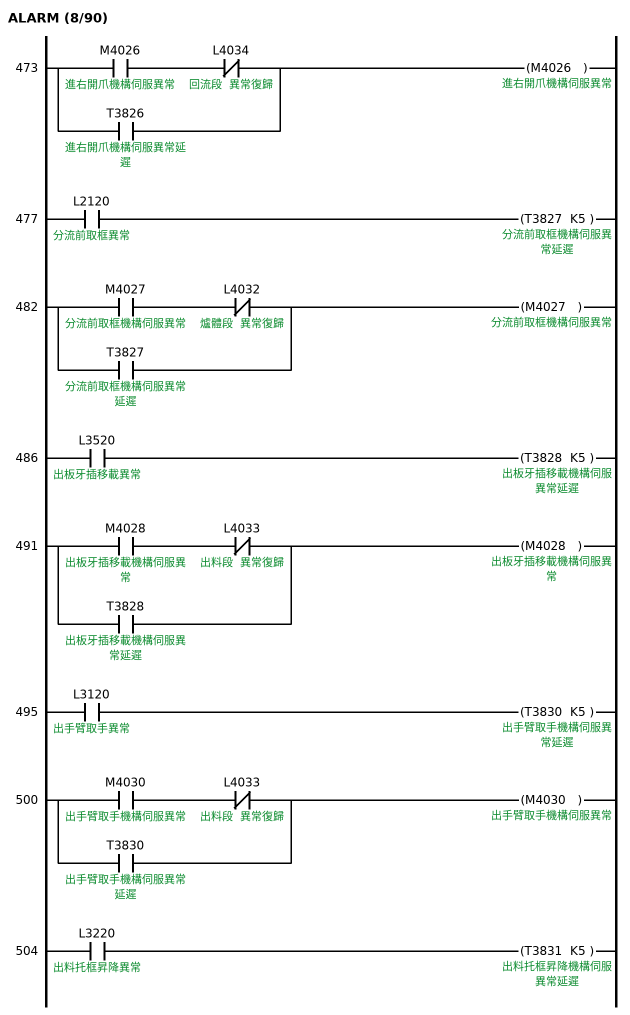
473   LD      M4026  ; 進右開爪機構伺服異常
      ANI     L4034  ; 回流段  異常復歸
      OR      T3826  ; 進右開爪機構伺服異常延遲
      OUT     M4026  ; 進右開爪機構伺服異常
477   LD      L2120  ; 分流前取框異常
      OUT     T3827 K5  ; 分流前取框機構伺服異常延遲
482   LD      M4027  ; 分流前取框機構伺服異常
      ANI     L4032  ; 爐體段  異常復歸
      OR      T3827  ; 分流前取框機構伺服異常延遲
      OUT     M4027  ; 分流前取框機構伺服異常
486   LD      L3520  ; 出板牙插移載異常
      OUT     T3828 K5  ; 出板牙插移載機構伺服異常延遲
491   LD      M4028  ; 出板牙插移載機構伺服異常
      ANI     L4033  ; 出料段  異常復歸
      OR      T3828  ; 出板牙插移載機構伺服異常延遲
      OUT     M4028  ; 出板牙插移載機構伺服異常
495   LD      L3120  ; 出手臂取手異常
      OUT     T3830 K5  ; 出手臂取手機構伺服異常延遲
500   LD      M4030  ; 出手臂取手機構伺服異常
      ANI     L4033  ; 出料段  異常復歸
      OR      T3830  ; 出手臂取手機構伺服異常延遲
      OUT     M4030  ; 出手臂取手機構伺服異常
504   LD      L3220  ; 出料托框昇降異常
      OUT     T3831 K5  ; 出料托框昇降機構伺服異常延遲
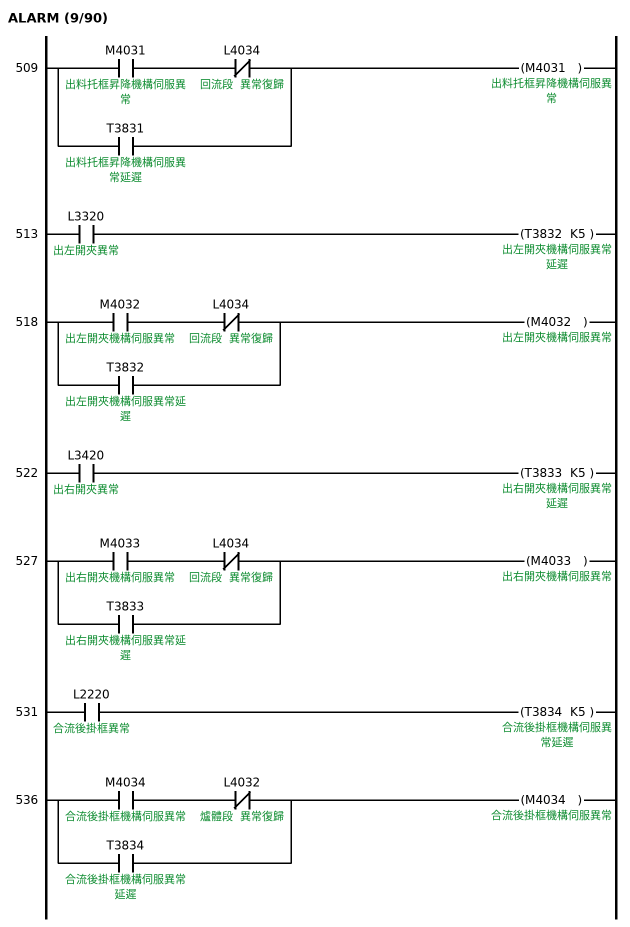
509   LD      M4031  ; 出料托框昇降機構伺服異常
      ANI     L4034  ; 回流段  異常復歸
      OR      T3831  ; 出料托框昇降機構伺服異常延遲
      OUT     M4031  ; 出料托框昇降機構伺服異常
513   LD      L3320  ; 出左開夾異常
      OUT     T3832 K5  ; 出左開夾機構伺服異常延遲
518   LD      M4032  ; 出左開夾機構伺服異常
      ANI     L4034  ; 回流段  異常復歸
      OR      T3832  ; 出左開夾機構伺服異常延遲
      OUT     M4032  ; 出左開夾機構伺服異常
522   LD      L3420  ; 出右開夾異常
      OUT     T3833 K5  ; 出右開夾機構伺服異常延遲
527   LD      M4033  ; 出右開夾機構伺服異常
      ANI     L4034  ; 回流段  異常復歸
      OR      T3833  ; 出右開夾機構伺服異常延遲
      OUT     M4033  ; 出右開夾機構伺服異常
531   LD      L2220  ; 合流後掛框異常
      OUT     T3834 K5  ; 合流後掛框機構伺服異常延遲
536   LD      M4034  ; 合流後掛框機構伺服異常
      ANI     L4032  ; 爐體段  異常復歸
      OR      T3834  ; 合流後掛框機構伺服異常延遲
      OUT     M4034  ; 合流後掛框機構伺服異常
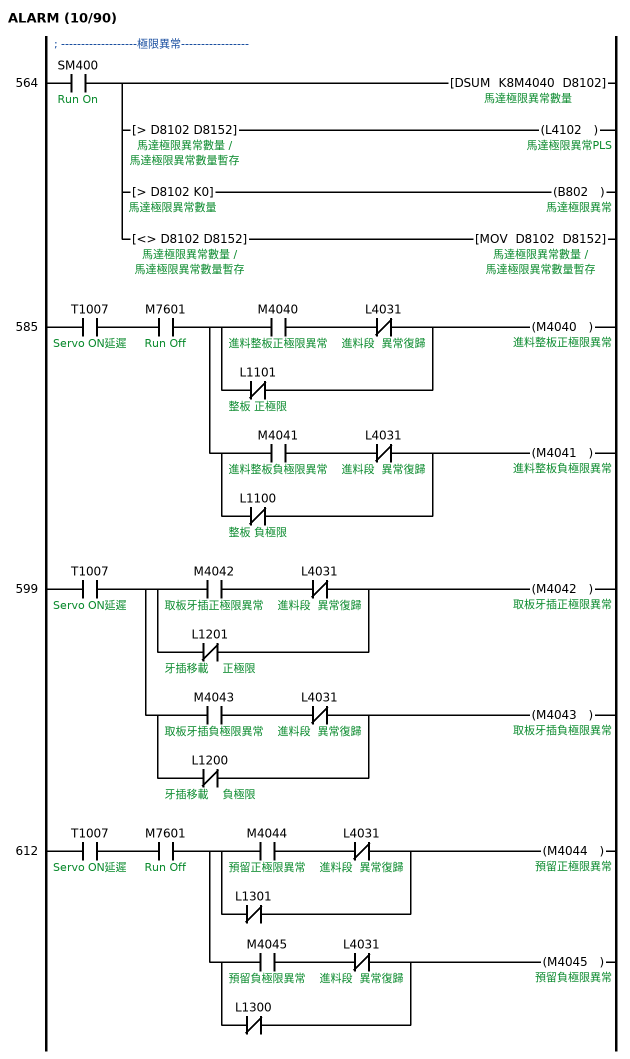
; -------------------極限異常-----------------
564   LD      SM400  ; Run On
      DSUM    K8M4040 D8102  ; 進料整板正極限異常 / 馬達極限異常數量
      MPS
      AND>    D8102 D8152  ; 馬達極限異常數量 / 馬達極限異常數量暫存
      OUT     L4102  ; 馬達極限異常PLS
      MRD
      AND>    D8102 K0  ; 馬達極限異常數量
      OUT     B802  ; 馬達極限異常
      MPP
      AND<>   D8102 D8152  ; 馬達極限異常數量 / 馬達極限異常數量暫存
      MOV     D8102 D8152
585   LD      T1007  ; Servo ON延遲
      AND     M7601  ; Run Off
      MPS
      LD      M4040  ; 進料整板正極限異常
      ANI     L4031  ; 進料段  異常復歸
      ORI     L1101  ; 整板 正極限
      ANB
      OUT     M4040  ; 進料整板正極限異常
      MPP
      LD      M4041  ; 進料整板負極限異常
      ANI     L4031  ; 進料段  異常復歸
      ORI     L1100  ; 整板 負極限
      ANB
      OUT     M4041  ; 進料整板負極限異常
599   LD      T1007  ; Servo ON延遲
      MPS
      LD      M4042  ; 取板牙插正極限異常
      ANI     L4031  ; 進料段  異常復歸
      ORI     L1201  ; 牙插移載    正極限
      ANB
      OUT     M4042  ; 取板牙插正極限異常
      MPP
      LD      M4043  ; 取板牙插負極限異常
      ANI     L4031  ; 進料段  異常復歸
      ORI     L1200  ; 牙插移載    負極限
      ANB
      OUT     M4043  ; 取板牙插負極限異常
612   LD      T1007  ; Servo ON延遲
      AND     M7601  ; Run Off
      MPS
      LD      M4044  ; 預留正極限異常
      ANI     L4031  ; 進料段  異常復歸
      ORI     L1301
      ANB
      OUT     M4044  ; 預留正極限異常
      MPP
      LD      M4045  ; 預留負極限異常
      ANI     L4031  ; 進料段  異常復歸
      ORI     L1300
      ANB
      OUT     M4045  ; 預留負極限異常
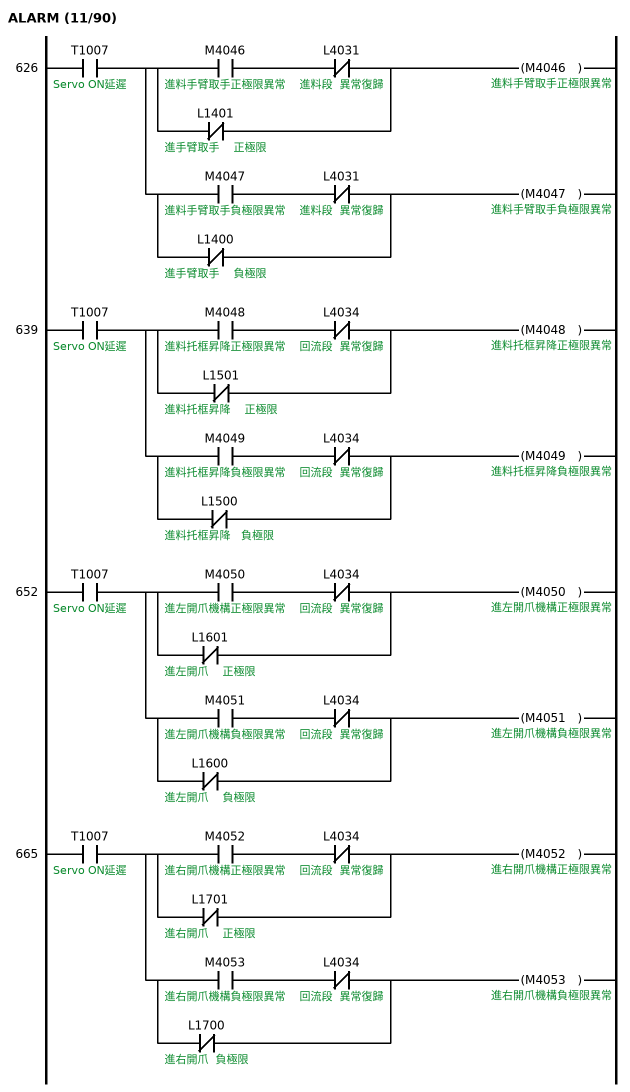
626   LD      T1007  ; Servo ON延遲
      MPS
      LD      M4046  ; 進料手臂取手正極限異常
      ANI     L4031  ; 進料段  異常復歸
      ORI     L1401  ; 進手臂取手    正極限
      ANB
      OUT     M4046  ; 進料手臂取手正極限異常
      MPP
      LD      M4047  ; 進料手臂取手負極限異常
      ANI     L4031  ; 進料段  異常復歸
      ORI     L1400  ; 進手臂取手    負極限
      ANB
      OUT     M4047  ; 進料手臂取手負極限異常
639   LD      T1007  ; Servo ON延遲
      MPS
      LD      M4048  ; 進料托框昇降正極限異常
      ANI     L4034  ; 回流段  異常復歸
      ORI     L1501  ; 進料托框昇降    正極限
      ANB
      OUT     M4048  ; 進料托框昇降正極限異常
      MPP
      LD      M4049  ; 進料托框昇降負極限異常
      ANI     L4034  ; 回流段  異常復歸
      ORI     L1500  ; 進料托框昇降   負極限
      ANB
      OUT     M4049  ; 進料托框昇降負極限異常
652   LD      T1007  ; Servo ON延遲
      MPS
      LD      M4050  ; 進左開爪機構正極限異常
      ANI     L4034  ; 回流段  異常復歸
      ORI     L1601  ; 進左開爪    正極限
      ANB
      OUT     M4050  ; 進左開爪機構正極限異常
      MPP
      LD      M4051  ; 進左開爪機構負極限異常
      ANI     L4034  ; 回流段  異常復歸
      ORI     L1600  ; 進左開爪    負極限
      ANB
      OUT     M4051  ; 進左開爪機構負極限異常
665   LD      T1007  ; Servo ON延遲
      MPS
      LD      M4052  ; 進右開爪機構正極限異常
      ANI     L4034  ; 回流段  異常復歸
      ORI     L1701  ; 進右開爪    正極限
      ANB
      OUT     M4052  ; 進右開爪機構正極限異常
      MPP
      LD      M4053  ; 進右開爪機構負極限異常
      ANI     L4034  ; 回流段  異常復歸
      ORI     L1700  ; 進右開爪  負極限
      ANB
      OUT     M4053  ; 進右開爪機構負極限異常
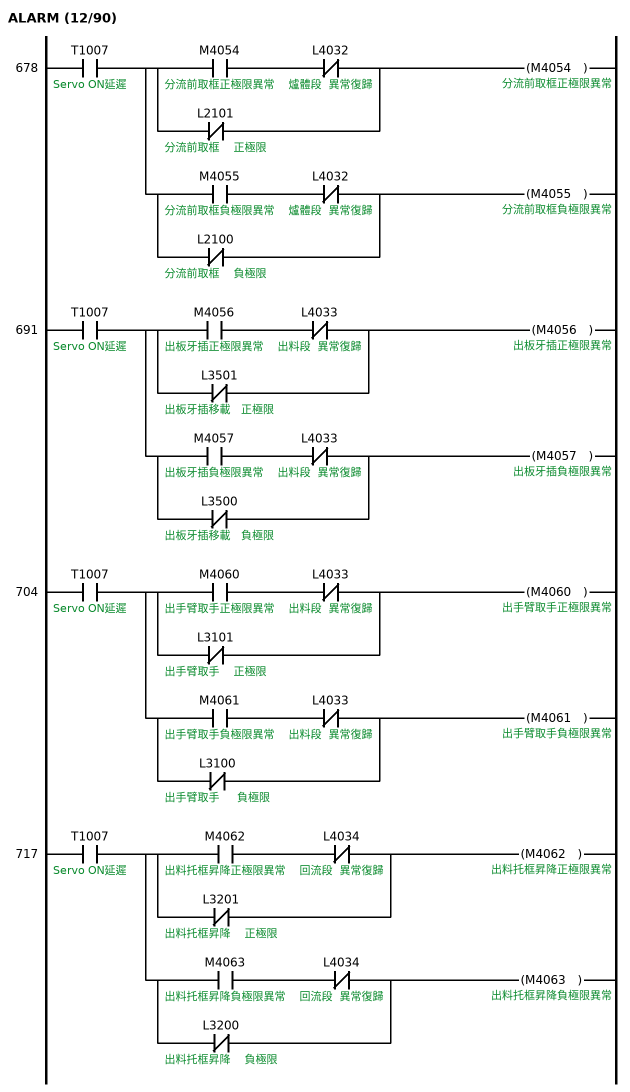
678   LD      T1007  ; Servo ON延遲
      MPS
      LD      M4054  ; 分流前取框正極限異常
      ANI     L4032  ; 爐體段  異常復歸
      ORI     L2101  ; 分流前取框    正極限
      ANB
      OUT     M4054  ; 分流前取框正極限異常
      MPP
      LD      M4055  ; 分流前取框負極限異常
      ANI     L4032  ; 爐體段  異常復歸
      ORI     L2100  ; 分流前取框    負極限
      ANB
      OUT     M4055  ; 分流前取框負極限異常
691   LD      T1007  ; Servo ON延遲
      MPS
      LD      M4056  ; 出板牙插正極限異常
      ANI     L4033  ; 出料段  異常復歸
      ORI     L3501  ; 出板牙插移載   正極限
      ANB
      OUT     M4056  ; 出板牙插正極限異常
      MPP
      LD      M4057  ; 出板牙插負極限異常
      ANI     L4033  ; 出料段  異常復歸
      ORI     L3500  ; 出板牙插移載   負極限
      ANB
      OUT     M4057  ; 出板牙插負極限異常
704   LD      T1007  ; Servo ON延遲
      MPS
      LD      M4060  ; 出手臂取手正極限異常
      ANI     L4033  ; 出料段  異常復歸
      ORI     L3101  ; 出手臂取手    正極限
      ANB
      OUT     M4060  ; 出手臂取手正極限異常
      MPP
      LD      M4061  ; 出手臂取手負極限異常
      ANI     L4033  ; 出料段  異常復歸
      ORI     L3100  ; 出手臂取手     負極限
      ANB
      OUT     M4061  ; 出手臂取手負極限異常
717   LD      T1007  ; Servo ON延遲
      MPS
      LD      M4062  ; 出料托框昇降正極限異常
      ANI     L4034  ; 回流段  異常復歸
      ORI     L3201  ; 出料托框昇降    正極限
      ANB
      OUT     M4062  ; 出料托框昇降正極限異常
      MPP
      LD      M4063  ; 出料托框昇降負極限異常
      ANI     L4034  ; 回流段  異常復歸
      ORI     L3200  ; 出料托框昇降    負極限
      ANB
      OUT     M4063  ; 出料托框昇降負極限異常
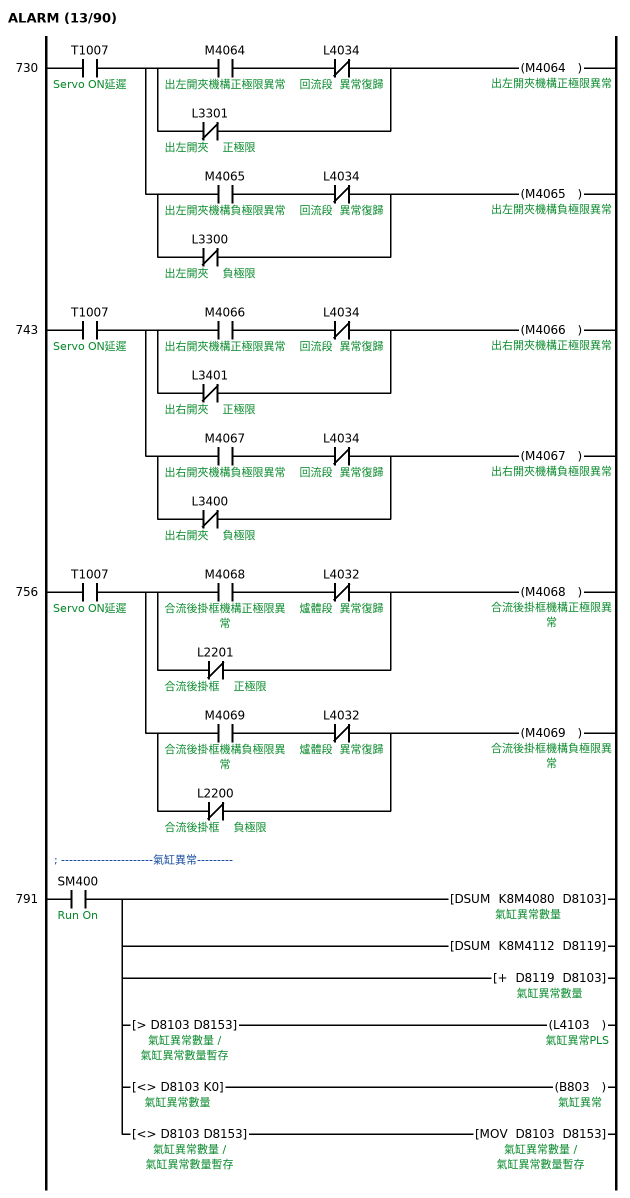
730   LD      T1007  ; Servo ON延遲
      MPS
      LD      M4064  ; 出左開夾機構正極限異常
      ANI     L4034  ; 回流段  異常復歸
      ORI     L3301  ; 出左開夾    正極限
      ANB
      OUT     M4064  ; 出左開夾機構正極限異常
      MPP
      LD      M4065  ; 出左開夾機構負極限異常
      ANI     L4034  ; 回流段  異常復歸
      ORI     L3300  ; 出左開夾    負極限
      ANB
      OUT     M4065  ; 出左開夾機構負極限異常
743   LD      T1007  ; Servo ON延遲
      MPS
      LD      M4066  ; 出右開夾機構正極限異常
      ANI     L4034  ; 回流段  異常復歸
      ORI     L3401  ; 出右開夾    正極限
      ANB
      OUT     M4066  ; 出右開夾機構正極限異常
      MPP
      LD      M4067  ; 出右開夾機構負極限異常
      ANI     L4034  ; 回流段  異常復歸
      ORI     L3400  ; 出右開夾    負極限
      ANB
      OUT     M4067  ; 出右開夾機構負極限異常
756   LD      T1007  ; Servo ON延遲
      MPS
      LD      M4068  ; 合流後掛框機構正極限異常
      ANI     L4032  ; 爐體段  異常復歸
      ORI     L2201  ; 合流後掛框    正極限
      ANB
      OUT     M4068  ; 合流後掛框機構正極限異常
      MPP
      LD      M4069  ; 合流後掛框機構負極限異常
      ANI     L4032  ; 爐體段  異常復歸
      ORI     L2200  ; 合流後掛框    負極限
      ANB
      OUT     M4069  ; 合流後掛框機構負極限異常
; -----------------------氣缸異常---------
791   LD      SM400  ; Run On
      DSUM    K8M4080 D8103  ; 進料牙叉上昇降異常 / 氣缸異常數量
      DSUM    K8M4112 D8119  ; 出料牙叉夾板氣缸夾異常
      +       D8119 D8103
      MPS
      AND>    D8103 D8153  ; 氣缸異常數量 / 氣缸異常數量暫存
      OUT     L4103  ; 氣缸異常PLS
      MRD
      AND<>   D8103 K0  ; 氣缸異常數量
      OUT     B803  ; 氣缸異常
      MPP
      AND<>   D8103 D8153  ; 氣缸異常數量 / 氣缸異常數量暫存
      MOV     D8103 D8153
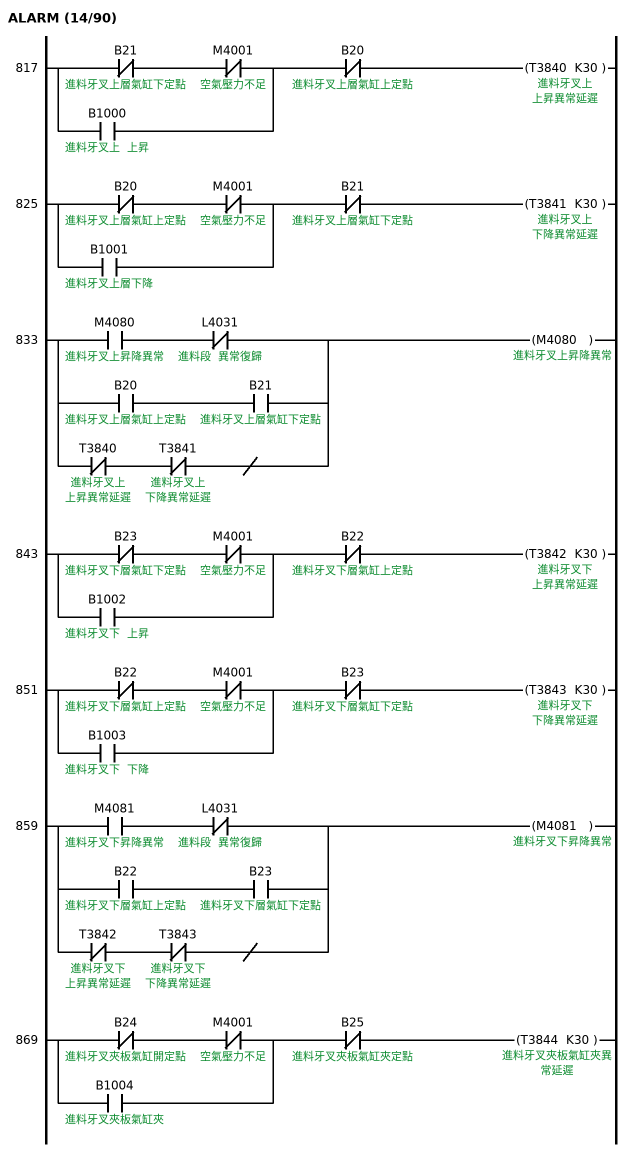
817   LDI     B21  ; 進料牙叉上層氣缸下定點
      ANI     M4001  ; 空氣壓力不足
      OR      B1000  ; 進料牙叉上  上昇
      ANI     B20  ; 進料牙叉上層氣缸上定點
      OUT     T3840 K30  ; 進料牙叉上  上昇異常延遲
825   LDI     B20  ; 進料牙叉上層氣缸上定點
      ANI     M4001  ; 空氣壓力不足
      OR      B1001  ; 進料牙叉上層下降
      ANI     B21  ; 進料牙叉上層氣缸下定點
      OUT     T3841 K30  ; 進料牙叉上  下降異常延遲
833   LD      M4080  ; 進料牙叉上昇降異常
      ANI     L4031  ; 進料段  異常復歸
      LD      B20  ; 進料牙叉上層氣缸上定點
      AND     B21  ; 進料牙叉上層氣缸下定點
      ORB
      LDI     T3840  ; 進料牙叉上  上昇異常延遲
      ANI     T3841  ; 進料牙叉上  下降異常延遲
      INV
      ORB
      OUT     M4080  ; 進料牙叉上昇降異常
843   LDI     B23  ; 進料牙叉下層氣缸下定點
      ANI     M4001  ; 空氣壓力不足
      OR      B1002  ; 進料牙叉下  上昇
      ANI     B22  ; 進料牙叉下層氣缸上定點
      OUT     T3842 K30  ; 進料牙叉下  上昇異常延遲
851   LDI     B22  ; 進料牙叉下層氣缸上定點
      ANI     M4001  ; 空氣壓力不足
      OR      B1003  ; 進料牙叉下  下降
      ANI     B23  ; 進料牙叉下層氣缸下定點
      OUT     T3843 K30  ; 進料牙叉下  下降異常延遲
859   LD      M4081  ; 進料牙叉下昇降異常
      ANI     L4031  ; 進料段  異常復歸
      LD      B22  ; 進料牙叉下層氣缸上定點
      AND     B23  ; 進料牙叉下層氣缸下定點
      ORB
      LDI     T3842  ; 進料牙叉下  上昇異常延遲
      ANI     T3843  ; 進料牙叉下  下降異常延遲
      INV
      ORB
      OUT     M4081  ; 進料牙叉下昇降異常
869   LDI     B24  ; 進料牙叉夾板氣缸開定點
      ANI     M4001  ; 空氣壓力不足
      OR      B1004  ; 進料牙叉夾板氣缸夾
      ANI     B25  ; 進料牙叉夾板氣缸夾定點
      OUT     T3844 K30  ; 進料牙叉夾板氣缸夾異常延遲
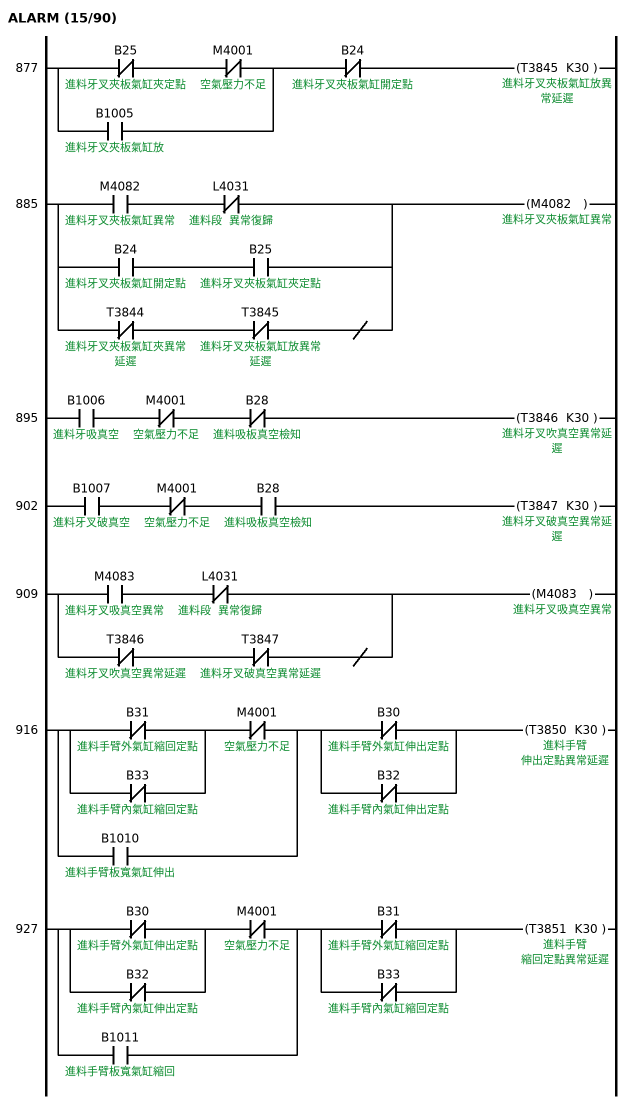
877   LDI     B25  ; 進料牙叉夾板氣缸夾定點
      ANI     M4001  ; 空氣壓力不足
      OR      B1005  ; 進料牙叉夾板氣缸放
      ANI     B24  ; 進料牙叉夾板氣缸開定點
      OUT     T3845 K30  ; 進料牙叉夾板氣缸放異常延遲
885   LD      M4082  ; 進料牙叉夾板氣缸異常
      ANI     L4031  ; 進料段  異常復歸
      LD      B24  ; 進料牙叉夾板氣缸開定點
      AND     B25  ; 進料牙叉夾板氣缸夾定點
      ORB
      LDI     T3844  ; 進料牙叉夾板氣缸夾異常延遲
      ANI     T3845  ; 進料牙叉夾板氣缸放異常延遲
      INV
      ORB
      OUT     M4082  ; 進料牙叉夾板氣缸異常
895   LD      B1006  ; 進料牙吸真空
      ANI     M4001  ; 空氣壓力不足
      ANI     B28  ; 進料吸板真空檢知
      OUT     T3846 K30  ; 進料牙叉吹真空異常延遲
902   LD      B1007  ; 進料牙叉破真空
      ANI     M4001  ; 空氣壓力不足
      AND     B28  ; 進料吸板真空檢知
      OUT     T3847 K30  ; 進料牙叉破真空異常延遲
909   LD      M4083  ; 進料牙叉吸真空異常
      ANI     L4031  ; 進料段  異常復歸
      LDI     T3846  ; 進料牙叉吹真空異常延遲
      ANI     T3847  ; 進料牙叉破真空異常延遲
      INV
      ORB
      OUT     M4083  ; 進料牙叉吸真空異常
916   LDI     B31  ; 進料手臂外氣缸縮回定點
      ORI     B33  ; 進料手臂內氣缸縮回定點
      ANI     M4001  ; 空氣壓力不足
      OR      B1010  ; 進料手臂板寬氣缸伸出
      LDI     B30  ; 進料手臂外氣缸伸出定點
      ORI     B32  ; 進料手臂內氣缸伸出定點
      ANB
      OUT     T3850 K30  ; 進料手臂   伸出定點異常延遲
927   LDI     B30  ; 進料手臂外氣缸伸出定點
      ORI     B32  ; 進料手臂內氣缸伸出定點
      ANI     M4001  ; 空氣壓力不足
      OR      B1011  ; 進料手臂板寬氣缸縮回
      LDI     B31  ; 進料手臂外氣缸縮回定點
      ORI     B33  ; 進料手臂內氣缸縮回定點
      ANB
      OUT     T3851 K30  ; 進料手臂   縮回定點異常延遲
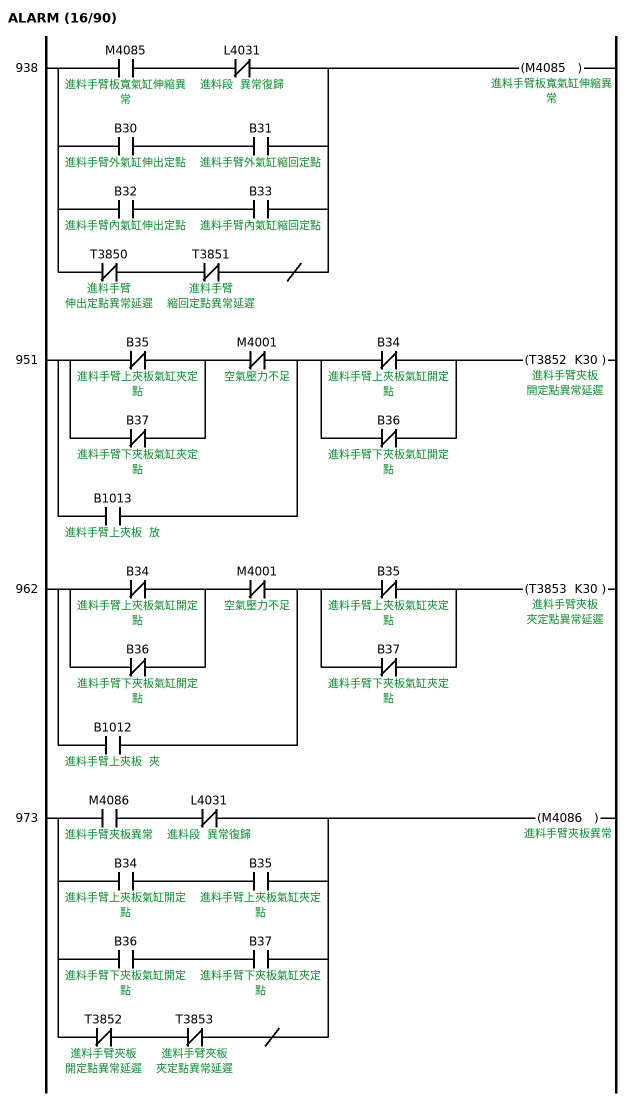
938   LD      M4085  ; 進料手臂板寬氣缸伸縮異常
      ANI     L4031  ; 進料段  異常復歸
      LD      B30  ; 進料手臂外氣缸伸出定點
      AND     B31  ; 進料手臂外氣缸縮回定點
      ORB
      LD      B32  ; 進料手臂內氣缸伸出定點
      AND     B33  ; 進料手臂內氣缸縮回定點
      ORB
      LDI     T3850  ; 進料手臂   伸出定點異常延遲
      ANI     T3851  ; 進料手臂   縮回定點異常延遲
      INV
      ORB
      OUT     M4085  ; 進料手臂板寬氣缸伸縮異常
951   LDI     B35  ; 進料手臂上夾板氣缸夾定點
      ORI     B37  ; 進料手臂下夾板氣缸夾定點
      ANI     M4001  ; 空氣壓力不足
      OR      B1013  ; 進料手臂上夾板  放
      LDI     B34  ; 進料手臂上夾板氣缸開定點
      ORI     B36  ; 進料手臂下夾板氣缸開定點
      ANB
      OUT     T3852 K30  ; 進料手臂夾板    開定點異常延遲
962   LDI     B34  ; 進料手臂上夾板氣缸開定點
      ORI     B36  ; 進料手臂下夾板氣缸開定點
      ANI     M4001  ; 空氣壓力不足
      OR      B1012  ; 進料手臂上夾板  夾
      LDI     B35  ; 進料手臂上夾板氣缸夾定點
      ORI     B37  ; 進料手臂下夾板氣缸夾定點
      ANB
      OUT     T3853 K30  ; 進料手臂夾板    夾定點異常延遲
973   LD      M4086  ; 進料手臂夾板異常
      ANI     L4031  ; 進料段  異常復歸
      LD      B34  ; 進料手臂上夾板氣缸開定點
      AND     B35  ; 進料手臂上夾板氣缸夾定點
      ORB
      LD      B36  ; 進料手臂下夾板氣缸開定點
      AND     B37  ; 進料手臂下夾板氣缸夾定點
      ORB
      LDI     T3852  ; 進料手臂夾板    開定點異常延遲
      ANI     T3853  ; 進料手臂夾板    夾定點異常延遲
      INV
      ORB
      OUT     M4086  ; 進料手臂夾板異常
